INTERFACE I_LinkedListNode EXTENDS I_Disposable

METHOD PUBLIC Destroy
VAR_INPUT
END_VAR
END_METHOD

METHOD PUBLIC Equals : BOOL
VAR_INPUT
	Symbol : ANY;
END_VAR
END_METHOD

METHOD PUBLIC Get : BOOL;
VAR_INPUT
	Destination : ANY;
END_VAR
END_METHOD

METHOD PUBLIC GetTo : BOOL;
VAR_INPUT
	Destination : PVOID;
	DestinationSize : UDINT;
END_VAR
END_METHOD

PROPERTY PUBLIC Next : I_LinkedListNode
GET
END_GET
SET
END_SET
END_PROPERTY

PROPERTY PUBLIC Previous : I_LinkedListNode
GET
END_GET
SET
END_SET
END_PROPERTY

END_INTERFACE

(* stored: Version 1.1.0.1, ProductVersion 3.1.4024.12
   Itf I_LinkedListNode: Id {0cff8fbe-58e6-42f0-93b9-bcbf9ae1547a}
   Method Destroy: Id {63a4bd84-b6d5-48f0-b124-677ef16e8f2b}
   Method Equals: Id {42524c8e-5be9-4ec1-9fd9-53150bfb09c1}
   Method Get: Id {3cf610bf-474c-45ea-8852-ef97d7e3e565}
   Method GetTo: Id {81368b44-2f37-4a7b-af91-c3727dbd41a7}
   Property Next: Id {36f7d60e-da19-4ec7-aef7-5f62014911e7}
   Get Get: Id {e871223f-e76e-40e1-ac6e-8232b4f33a89}
   Set Set: Id {01642d6e-14c4-4289-a99f-8469c57d0bae}
   Property Previous: Id {391f15bb-7210-4ad5-9151-9a7de912f823}
   Get Get: Id {855706cd-3426-4a83-93fc-01ff73e63b41}
   Set Set: Id {d562e515-c3b0-4344-956f-865d275d909b} *)
